// TIA Portal V21 export
TYPE "lubricationSystemAlm"
   STRUCT
      stepErr : Bool;
      noPumpSelected : Bool;
      pump1Fault : Bool;
      pump2Fault : Bool;
      lowOilLevel : Bool;
      lowOilTempTankSw : Bool;   // Low oil temperature in tank switch
      highOilTempTankSw : Bool;   // High oil temperature in tank switch
      extStop : Bool;
      unableToEstablishFlow : Bool;
      noReturnOilFlow : Bool;
      unableToDisablePumps : Bool;
      badHeaterCoolerParams : Bool;   // Heater and cooler setpoints overlap
      oilTempTankHiHi : Bool;
      oilTempTankLoLo : Bool;
      lowOilFlow : Bool;
   END_STRUCT;
END_TYPE
